GLOBALCONSTANTS DefaultPool (* Global constants *)
  VAR_GLOBAL CONSTANT
    ISO_DESIGNATOR_WIDTH : UINT := 80;
    ISO_DESIGNATOR_HEIGHT : UINT := 80;
    ISO_MASK_SIZE : UINT := 480;
    ISO_VERSION_LABEL : STRING;
    MASK_WIDTH : UINT := 480;
    MASK_HEIGHT : UINT := 480;
    WorkingSet_0 : UINT := 0;
    DataMask_1000 : UINT := 1000;
    SoftKeyMask_PAGE_1 : UINT := 4000;
    SoftKeyMask_PAGE_2 : UINT := 4001;
    SoftKey_Automatik_ein : UINT := 5000;
    SoftKey_Dom : UINT := 5001;
    SoftKey_Heckschieber : UINT := 5002;
    SoftKey_Auseinanderklappen : UINT := 5003;
    SoftKey_Verteiler_senken : UINT := 5004;
    SoftKey_Knickdeichsel_senken : UINT := 5005;
    SoftKey_Automatik_aus : UINT := 5006;
    SoftKey_Schneidwerk : UINT := 5007;
    SoftKey_Seitenschieber : UINT := 5008;
    SoftKey_Zusammenklappen : UINT := 5009;
    SoftKey_Verteiler_heben : UINT := 5010;
    SoftKey_Knickdeichsel_heben : UINT := 5011;
    SoftKey_5012 : UINT := 5012;
    SoftKey_5013 : UINT := 5013;
    SoftKey_Abscheider : UINT := 5015;
    SoftKey_Licht : UINT := 5016;
    SoftKey_5017 : UINT := 5017;
    SoftKey_5018 : UINT := 5018;
    SoftKey_5019 : UINT := 5019;
    SoftKey_5021 : UINT := 5021;
    SoftKey_5022 : UINT := 5022;
    SoftKey_5023 : UINT := 5023;
    PAGE_1_BTN : UINT := 6000;
    PAGE_2_BTN : UINT := 6001;
    page_2_MAIN : UINT := 20002;
    page_1_MAIN : UINT := 20003;
    workingset_pic : UINT := 20500;
    Automatik_ein : UINT := 20501;
    Automatik_aus : UINT := 20502;
    Einfuelldom : UINT := 20503;
    EXACUT : UINT := 20504;
    Seitenschieber : UINT := 20505;
    Heckschieber : UINT := 20506;
    zusammenklappen : UINT := 20507;
    auseinanderklappen : UINT := 20508;
    Verteiler_heben : UINT := 20509;
    Verteiler_senken : UINT := 20510;
    Knickdeichsel_heben : UINT := 20511;
    Knickdeichsel_senken : UINT := 20512;
    lightbulb : UINT := 20513;
    trash_icon : UINT := 20514;
    page_1_for_AUX : UINT := 20516;
    page_2_for_AUX : UINT := 20517;
    AuxInput_Automatik_ein : UINT := 31000;
    AuxInput_Dom : UINT := 31001;
    AuxInput_Heckschieber : UINT := 31002;
    AuxInput_Auseinanderklappen : UINT := 31003;
    AuxInput_Verteiler_senken : UINT := 31004;
    AuxInput_Knickdeichsel_senken : UINT := 31005;
    AuxInput_Automatik_aus : UINT := 31006;
    AuxInput_Schneidwerk : UINT := 31007;
    AuxInput_Seitenschieber : UINT := 31008;
    AuxInput_Zusammenklappen : UINT := 31009;
    AuxInput_Verteiler_heben : UINT := 31010;
    AuxInput_Knickdeichsel_heben : UINT := 31011;
    AuxInput_Abscheider : UINT := 31015;
    AuxInput_Licht : UINT := 31016;
    PAGE_1_AUX : UINT := 31024;
    PAGE_2_AUX : UINT := 31025;
  END_VAR
END_GLOBALCONSTANTS
